SUBAPPLICATION AX_SoftkeySR_TO_QXA_BG (* 3 Softkeys (SET/RESET/TOGGLE) auf AX_T_FF_SR, Ausgang QXA + Background (am TOGGLE-Key). Generisch. *)
  (* Standard: 61499-2 *)
  (* Version 1.0, 2026-09-09, Franz Höpfinger, Meisterschulen am Ostbahnhof, Ausgelagert aus Uebung_010e2_sub_AX zur Wiederverwendung; u16ObjId_SET/_RESET/_TOGGLE und Output zuvor fest importiert (SoftKey_F1/F2/F3, Output_Q1), jetzt generische Defaults (ID_NULL/Invalid). *)
  PACKAGE MyLib::sys;
  IMPORT isobus::UT::Q::const::IDs::ID_NULL;
  IMPORT logiBUS::io::DQ::logiBUS_DO;
  IMPORT logiBUS::io::DQ::logiBUS_DO_S;
  IMPORT isobus::UT::io::Softkey::SoftKeyActivationCode::SK_RELEASED;
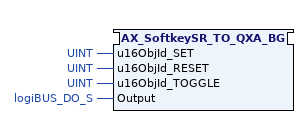
  VAR_INPUT
    u16ObjId_SET : UINT := ID_NULL; (* Object ID SET SoftKey *)
    u16ObjId_RESET : UINT := ID_NULL; (* Object ID RESET SoftKey *)
    u16ObjId_TOGGLE : UINT := ID_NULL; (* Object ID TOGGLE SoftKey (auch fuer GreenWhiteBackground) *)
    Output : logiBUS::io::DQ::logiBUS_DO_S := logiBUS_DO::Invalid; (* Identify the Output Output_Q1..Q8 *)
  END_VAR
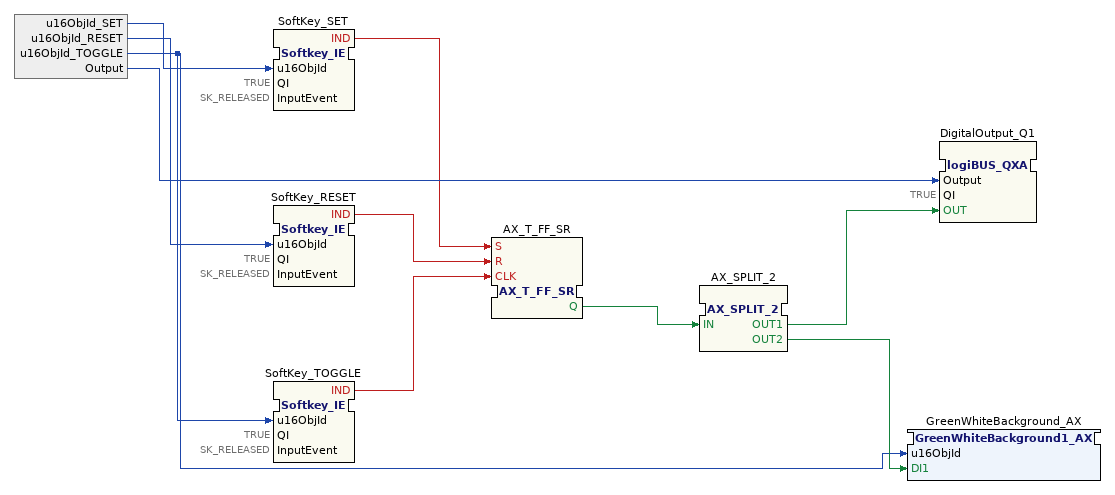
  FBS
    SoftKey_SET : isobus::UT::io::Softkey::Softkey_IE(QI := TRUE, InputEvent := SK_RELEASED);
    SoftKey_RESET : isobus::UT::io::Softkey::Softkey_IE(QI := TRUE, InputEvent := SK_RELEASED);
    SoftKey_TOGGLE : isobus::UT::io::Softkey::Softkey_IE(QI := TRUE, InputEvent := SK_RELEASED);
    AX_T_FF_SR : adapter::events::unidirectional::AX_T_FF_SR;
    AX_SPLIT_2 : adapter::events::unidirectional::AX_SPLIT_2;
    DigitalOutput_Q1 : logiBUS::io::DQ::logiBUS_QXA(QI := TRUE);
  END_FBS
  SUBAPPS
    GreenWhiteBackground_AX : MyLib::sys::GreenWhiteBackground1_AX;
  END_SUBAPPS
  EVENT_CONNECTIONS
    SoftKey_SET.IND TO AX_T_FF_SR.S;
    SoftKey_RESET.IND TO AX_T_FF_SR.R;
    SoftKey_TOGGLE.IND TO AX_T_FF_SR.CLK;
  END_CONNECTIONS
  DATA_CONNECTIONS
    u16ObjId_SET TO SoftKey_SET.u16ObjId;
    u16ObjId_RESET TO SoftKey_RESET.u16ObjId;
    u16ObjId_TOGGLE TO SoftKey_TOGGLE.u16ObjId;
    u16ObjId_TOGGLE TO GreenWhiteBackground_AX.u16ObjId;
    Output TO DigitalOutput_Q1.Output;
  END_CONNECTIONS
  ADAPTER_CONNECTIONS
    AX_T_FF_SR.Q TO AX_SPLIT_2.IN;
    AX_SPLIT_2.OUT1 TO DigitalOutput_Q1.OUT;
    AX_SPLIT_2.OUT2 TO GreenWhiteBackground_AX.DI1;
  END_CONNECTIONS
END_SUBAPPLICATION
